FUNCTION_BLOCK FB_AlarmHandler
VAR
	  bActive   : BOOL   := FALSE;
      sMessage  : STRING := '';
      tonBlink  : TON;
      bLampState: BOOL   := FALSE;
END_VAR

tonBlink(IN := bActive, PT := GVL_Constants.ALARM_BLINK);

IF tonBlink.Q THEN
    bLampState        := NOT bLampState;
    tonBlink(IN := FALSE, PT := GVL_Constants.ALARM_BLINK);
    tonBlink(IN := TRUE,  PT := GVL_Constants.ALARM_BLINK);
END_IF

GVL_IO.bAlarmLamp  := bActive AND bLampState;
GVL_IO.sAlarmMsg   := sMessage;

METHOD ClearAlarm : BOOL
VAR_INPUT
END_VAR
 bActive   := FALSE;
 sMessage  := '';
 bLampState:= FALSE;
 GVL_IO.bAlarmLamp := FALSE;
END_METHOD

PROPERTY IsActive : BOOL
GET
IsActive := bActive;
END_GET
SET
END_SET
END_PROPERTY

PROPERTY Message : STRING
GET
Message := sMessage;
END_GET
SET
END_SET
END_PROPERTY

METHOD SetAlarm : BOOL
VAR_INPUT
	sMsg : STRING;
END_VAR
bActive  := TRUE;
sMessage := sMsg;
END_METHOD

END_FUNCTION_BLOCK

(* stored: Version 1.1.0.1, ProductVersion 3.1.4024.16
   POU FB_AlarmHandler: Id {048ed448-ae4b-4070-8f07-f8008abbe27d}, SpecialFunc None
   Method ClearAlarm: Id {f6aa93e6-7af7-4737-97d7-ba64ba17d6ca}
   Property IsActive: Id {ccc025b8-8e0e-4e97-80d4-350d784ce4fc}
   Get Get: Id {4e02c545-b9bd-495a-9495-18a245a26bbd}
   Set Set: Id {96408d8f-a00b-4ec3-bec1-62d875f9ed00}
   Property Message: Id {c9bddd77-eeab-4f31-afa6-1d4aaea1a8fa}
   Get Get: Id {ebdd30fd-6652-44b3-b835-7dfdb686c2ff}
   Set Set: Id {82bbe2dd-f29f-437e-8f26-ad6e94d2dd29}
   Method SetAlarm: Id {cd065b06-f720-47e5-8a8d-1454ed7a154b} *)
